// TwinCAT 3 PLC project _14_Facade
// ProgramVersion: 3.1.4023.0
// libraries:
//   Tc2_MC2, * (Beckhoff Automation GmbH)
//   Tc2_Standard, * (Beckhoff Automation GmbH)
//   Tc2_System, * (Beckhoff Automation GmbH)
//   Tc3_Module, * (Beckhoff Automation GmbH)
// project tree:
//   Facade/ MC_Axis.TcPOU
//   / MAIN.TcPOU, PlcTask.TcTTO
// (motion and I/O tree: see PLC project 13_decorator)
// real-time tasks:
//   TASK PlcTask: cycle T#10ms, priority 20, ADS port 350
// variable links:

CONFIGURATION _14_Facade
    RESOURCE PLC ON TwinCAT3
        TASK PlcTask(INTERVAL := T#10ms, PRIORITY := 20);
        PROGRAM MAIN WITH PlcTask : MAIN;
    END_RESOURCE
END_CONFIGURATION

// ---- MAIN.TcPOU
PROGRAM MAIN
VAR
	axisControl					: MC_Axis;
	resetEnable					: BOOL;
END_VAR

(* 
	GOF 		Provide a unified interface to a set of interfaces in a subsystem. 
				Facade defines a higher-level interface that makes the subsystem easier to use.
*)
axisControl.cyclicUpdate();
IF resetEnable	THEN
	resetEnable := NOT axisControl.resetEnable();
END_IF

END_PROGRAM

// ---- Facade/MC_Axis.TcPOU
FUNCTION_BLOCK MC_Axis
(* PLCopen motion control statemachine states: 
   https://infosys.beckhoff.com/english.php?content=../content/1033/tcplclib_tc2_mc2/70041995.html&id=6831501888106392354
	   MCSTATE_UNDEFINED,
	   MCSTATE_DISABLED,
	   MCSTATE_STANDSTILL,
	   MCSTATE_ERRORSTOP,
	   MCSTATE_STOPPING,
	   MCSTATE_HOMING,
	   MCSTATE_DISCRETEMOTION,
	   MCSTATE_CONTINOUSMOTION,
	   MCSTATE_SYNCHRONIZEDMOTION
*)
VAR	
	_axis					: axis_ref;		

	// MC_Power
	mcPower					: MC_Power;
	mcReset					: MC_Reset;
	mcHalt					: MC_Halt;
	
	// Internals
	state					: INT;
	toggle					: BYTE;	
END_VAR

//*********************************************************
// Code implementation only in CyclicUpdate() method for consistency with templates
// enables the use of the interface
// but calling this base method can be used to pass IN_OUTs to the instance
// without calling any code in the instance
//*********************************************************
cyclicUpdate();

// Let's (mis-)use the default MC2 Motion states
// When using the MC2 defined states, the method cannot lock up the _axis block
// There is always a defined state that can be used by the other methods
(* https://infosys.beckhoff.com/english.php?content=../content/1033/tcplclib_tc2_mc2/70041995.html&id=6831501888106392354
   MC__axisSTATE_UNDEFINED,
   MC__axisSTATE_DISABLED,
   MC__axisSTATE_STANDSTILL,
   MC__axisSTATE_ERRORSTOP,
   MC__axisSTATE_STOPPING,
   MC__axisSTATE_HOMING,
   MC__axisSTATE_DISCRETEMOTION,
   MC__axisSTATE_CONTINOUSMOTION,
   MC__axisSTATE_SYNCHRONIZEDMOTION
*)
METHOD abort				: BOOL
// 
abort:=FALSE;

// Trigger the abort message
//M_sendRegisteredMessageWithPathAndArg(rT.Q AND _Log, sDevName, TC_EVENTS.EventClass__axis.msg_axis_Aborting, _axis.NcToPlc._axisId); 
mcPower.Enable						:= FALSE;

// Act depending on the motion state
CASE _axis.Status.MotionState OF
	MC_axisSTATE_UNDEFINED:				// Let's hope not ;)
		abort:=FALSE;					// No defined path here
			
	MC_axisSTATE_DISABLED:				// The desired end state
		abort:=TRUE;
		
	MC_axisSTATE_STANDSTILL:			// _axis is stopped, now disable it
		mcPower.Enable				:= FALSE;
		mcPower.Enable_Negative		:= FALSE;
		mcPower.Enable_Positive		:= FALSE;
		abort						:= FALSE;
		
	MC_axisSTATE_ERRORSTOP:				// Faulty end state, but it is an end state
		mcPower.Enable				:= FALSE;
		mcPower.Enable_Negative		:= FALSE;
		mcPower.Enable_Positive		:= FALSE;		
		abort						:= TRUE;
		
	MC_axisSTATE_STOPPING:				// intermediate state, nothing to do here
		mcPower.Enable				:= FALSE;
		mcPower.Enable_Negative		:= FALSE;
		mcPower.Enable_Positive		:= FALSE;
		abort						:= FALSE;
	
	// The _axis is still moving, first stop it
	MC_axisSTATE_HOMING,
	MC_axisSTATE_DISCRETEMOTION,
	MC_axisSTATE_CONTINOUSMOTION,
	MC_axisSTATE_SYNCHRONIZEDMOTION:
		mcPower.Enable				:= FALSE;
		mcPower.Enable_Negative		:= FALSE;
		mcPower.Enable_Positive		:= FALSE;
		abort						:= FALSE;
			
END_CASE
END_METHOD

PROPERTY PUBLIC axis : reference to axis_ref
GET
axis ref= _axis;
END_GET
END_PROPERTY

METHOD cyclicUpdate
VAR_INPUT
END_VAR
toggle	:= toggle + 1;

// Fetch _axis statusses
axis.ReadStatus();

// A_axiscontrol blocks
mcPower(
	axis			:= _axis, 
	Override			:= 100.0
	);
mcReset(axis:= _axis);
mcHalt(axis:= _axis);	
	
// Reset signals to function blocks, they will be re-set by the methods if necessary
mcHalt.Execute			:= FALSE;
mcReset.Execute			:= FALSE;
END_METHOD

METHOD reset		: BOOL
VAR_INPUT
END_VAR
// 
reset							:= FALSE;
mcHalt.Execute					:= FALSE;

// Act depending on the motion state
CASE _Axis.Status.MotionState OF
	MC_AXISSTATE_UNDEFINED:				// Let's hope not ;)
		reset:=FALSE;					// No defined path here
		
	MC_AXISSTATE_DISABLED,
	MC_AXISSTATE_STANDSTILL,			// The desired end state
	MC_AXISSTATE_SYNCHRONIZEDMOTION,
	MC_AXISSTATE_STOPPING,				
	MC_AXISSTATE_HOMING,
	MC_AXISSTATE_DISCRETEMOTION,
	MC_AXISSTATE_CONTINOUSMOTION:
		// DONKEY , TEMP HASJOB SOLUTION FOR KINEMATICS	
		IF _axis.Status.HasJob	OR _axis.Status.error 	THEN	// Try again, but leave the axis enabled
			mcReset.Execute		:= NOT mcReset.Execute AND toggle.3;
		ELSE
			reset:=TRUE;			// No defined path here
			mcReset.Execute			:= FALSE;
		END_IF
	
	MC_AXISSTATE_ERRORSTOP:				// Reset is necessary
		mcPower.Enable		:= FALSE;
		mcReset.Execute		:= NOT mcReset.Execute AND toggle.3;
		
END_CASE

// Reset OK
reset := NOT _axis.Status.Error AND NOT _axis.Status.HasJob;		// DONKEY , TEMP HASJOB SOLUTION FOR KINEMATICS
END_METHOD

METHOD resetEnable		: BOOL
VAR_INPUT
END_VAR
// 
resetEnable					:= FALSE;
mcHalt.Execute					:= FALSE;

// Act depending on the motion state
CASE _Axis.Status.MotionState OF
	MC_AXISSTATE_UNDEFINED:				// Let's hope not ;)
		resetEnable:=FALSE;					// No defined path here
		
	MC_AXISSTATE_DISABLED:				// Once the axis is disabled, start re-enabling it
		// Possibly transition from MC_AXISSTATE_ERRORSTOP
		// Pass parameters to Motion function
		mcPower.Enable			:= TRUE; 
		mcPower.Enable_Positive	:= TRUE; 
		mcPower.Enable_Negative	:= TRUE; 
		IF mcPower.Error		OR _axis.Status.error 	THEN		// try again 
			mcReset.Execute		:= NOT mcReset.Execute AND toggle.3;
			mcPower.Enable		:= FALSE; 
		END_IF
				
	MC_AXISSTATE_STANDSTILL,			// The desired end state
	MC_AXISSTATE_SYNCHRONIZEDMOTION:
		;
	
	MC_AXISSTATE_ERRORSTOP:				// Reset is necessary
		mcPower.Enable		:= FALSE;
		mcReset.Execute		:= NOT mcReset.Execute AND toggle.3;

	// Other states are to be ignored, disable all commands here			
	MC_AXISSTATE_STOPPING,				
	MC_AXISSTATE_HOMING,
	MC_AXISSTATE_DISCRETEMOTION,
	MC_AXISSTATE_CONTINOUSMOTION:
		// DONKEY , TEMP HASJOB SOLUTION FOR KINEMATICS	
		IF _axis.Status.HasJob	OR _axis.Status.error 	THEN	// Try again, but leave the axis enabled
			mcReset.Execute		:= NOT mcReset.Execute AND toggle.3;
		ELSE
			mcReset.Execute			:= FALSE;
		END_IF
		mcHalt.Execute				:= FALSE;
		
END_CASE

// Reset OK
resetEnable := mcPower.Status AND NOT _axis.Status.HasJob;		// DONKEY , TEMP HASJOB SOLUTION FOR KINEMATICS
END_METHOD

PROPERTY stateCurrent : MC_AxisStates
GET
StateCurrent := _axis.Status.MotionState;
END_GET
END_PROPERTY

// Let's (mis-)use the default MC2 Motion states
// When using the MC2 defined states, the method cannot lock up the axis block
// There is always a defined state that can be used by the other methods
(* https://infosys.beckhoff.com/english.php?content=../content/1033/tcplclib_tc2_mc2/70041995.html&id=6831501888106392354
   MC_AXISSTATE_UNDEFINED,
   MC_AXISSTATE_DISABLED,
   MC_AXISSTATE_STANDSTILL,
   MC_AXISSTATE_ERRORSTOP,
   MC_AXISSTATE_STOPPING,
   MC_AXISSTATE_HOMING,
   MC_AXISSTATE_DISCRETEMOTION,
   MC_AXISSTATE_CONTINOUSMOTION,
   MC_AXISSTATE_SYNCHRONIZEDMOTION
*)
METHOD stop				: BOOL
// 
stop:=FALSE;

// Act depending on the motion state
CASE _Axis.Status.MotionState OF
	MC_AXISSTATE_UNDEFINED:				// Let's hope not ;)
		stop:=FALSE;					// No defined path here
					
	MC_AXISSTATE_STANDSTILL,			// Axis is stopped, correct end state
	MC_AXISSTATE_DISABLED,				// Faulty end state, but it is an end state
	MC_AXISSTATE_ERRORSTOP:				// Faulty end state, but it is an end state
		mcHalt.Execute				:= FALSE;
		mcPower.Enable				:= FALSE;
		stop						:= TRUE;

	MC_AXISSTATE_STOPPING:				// intermediate state, nothing to do here
		stop						:= FALSE;
		
	// The axis is still moving, first stop it
	MC_AXISSTATE_HOMING,
	MC_AXISSTATE_DISCRETEMOTION,
	MC_AXISSTATE_CONTINOUSMOTION,
	MC_AXISSTATE_SYNCHRONIZEDMOTION:
		mcHalt.Execute				:= NOT mcHalt.Execute;	// Start to stop
		stop						:= FALSE;
					
END_CASE
END_METHOD

END_FUNCTION_BLOCK
